FUNCTION_BLOCK Q_ExecuteMacro (* Command Execute Macro( Part 6 - F.48 ) *)
  (* Standard: ISO 11783-6; Description: This message is available in VT Version 4 and later. This command is used to execute a Macro. Return values iso_s16 - E_NO_ERR - OK - E_OVERFLOW - buffer overflow - E_NOACT - Command not possible in current state - E_NO_INSTANCE - No VT client available *)
  (* Version 1.0, 2022-07-08, franz *)
  (* Documentation:
  This message is available in VT Version 4 and later. This command is used to execute a Macro.
   Return values
   iso_s16
    - E_NO_ERR - OK
   - E_OVERFLOW - buffer overflow
   - E_NOACT - Command not possible in current state
   - E_NO_INSTANCE - No VT client available
  *)
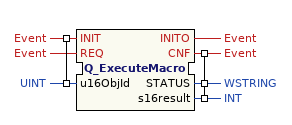
  EVENT_INPUT
    INIT WITH u16ObjId; (* Service Initialization *)
    REQ; (* Service Request *)
  END_EVENT
  EVENT_OUTPUT
    INITO; (* Initialization Confirm *)
    CNF WITH STATUS, s16result; (* Confirmation of Requested Service *)
  END_EVENT
  VAR_INPUT
    u16ObjId : UINT; (* Object ID of Macro object ( max. value 255 ) *)
  END_VAR
  VAR_OUTPUT
    STATUS : WSTRING; (* Service Status *)
    s16result : INT; (* retval see description *)
  END_VAR
END_FUNCTION_BLOCK
